FUNCTION_BLOCK FB_CartPowerOff EXTENDS FB_CartCtrlBase
VAR_INPUT
END_VAR
VAR_OUTPUT
END_VAR
VAR
	//output support leg break IO
	m_supportLegBreak :ARRAY [1..2] OF  DINT;
	
	// time threshold to 5-8joint after it's enabled
	m_cartAdjustStartWaitTime :LREAL := 0.2;
	
	//adjust start  time 
	m_adjustStartTime :LREAL;
END_VAR

// override this function in each exact controller
METHOD PROTECTED calcCmdJntPos : BOOL
VAR_IN_OUT CONSTANT
	// slave cart joint data
	i_slaveCart :FB_SlaveCart;
END_VAR

VAR
	i:INT;
END_VAR
//In this method, 8 represents the overhang angle
m_adjustStartTime :=LIMIT(0, m_adjustStartTime + g_cartCtrlCycleTime, 2);

m_isFinished :=supportLegUp(i_slaveCart );
END_METHOD

// override this function in each exact controller
// NOTICE: set joint control mode here, and do some initialization if needed
METHOD PUBLIC init : BOOL
VAR_IN_OUT CONSTANT
	i_slaveCart	:FB_SlaveCart;
END_VAR
VAR_IN_OUT 
	r_cartCtrlCmd :ST_SlaveArmCtrlCmds;
END_VAR
VAR
	i:INT;
END_VAR
//m_holdLastCmds := checkToHoldLastCmds(i_slaveCart);
m_holdLastCmds := checkToHoldLastCmds(i_slaveCart);

SUPER^.init(i_slaveCart,r_cartCtrlCmd);

m_jntEnableFlag[1] :=1;
m_jntEnableFlag[2] :=1;

m_jntOPMode[1]:= DriverOPMode_Trq;
m_jntOPMode[2]:= DriverOPMode_Trq;	

m_adjustStartTime := 0;
// update commands to arm
copyCmds(r_cartCtrlCmd);
END_METHOD

PROPERTY supportLegBreak : ARRAY [1..2] OF DINT
GET
supportLegBreak := m_supportLegBreak;
END_GET
END_PROPERTY

METHOD supportLegUp : BOOL
VAR_IN_OUT CONSTANT
	// slave cart joint data
	i_slaveCart :FB_SlaveCart;
END_VAR
VAR
	i : INT;
END_VAR

m_supportLegBreak[1] := 0;
m_supportLegBreak[2] := 0;

IF m_adjustStartTime > m_cartAdjustStartWaitTime THEN
	FOR i:=1 TO 2 DO
		m_cmdJntTrq[i] := 500;
	END_FOR
	
	IF NOT (i_slaveCart.m_supportLegSensor[1] OR i_slaveCart.m_supportLegSensor[2]) THEN
		supportLegUp := TRUE;
	END_IF
END_IF
END_METHOD

END_FUNCTION_BLOCK

(* stored: Version 1.1.0.1, ProductVersion 3.1.4024.11
   POU FB_CartPowerOff: Id {b2454179-7ec7-4ec5-8f34-e97cd4af4dc7}, SpecialFunc None
   Method calcCmdJntPos: Id {815a29ea-6288-402c-8876-55286ad97a38}
   Method init: Id {38f0555f-5b60-46bf-a5ad-9de6adcb181b}
   Property supportLegBreak: Id {621b1375-7d5a-434f-8b7a-bb65581340cf}
   Get Get: Id {cc2ce868-d9c6-4943-9361-d1a75a4ed62b}
   Method supportLegUp: Id {44d8502b-312d-4feb-9a41-704ba81e21d3} *)
